FUNCTION_BLOCK FB_Transfo_Base
//////////////////
// High Voltage transformer with Transfo or DMCR detection . 
//////////////////

VAR_INPUT PERSISTENT
	// Parameters of the Object (instance/model specific) 

END_VAR

VAR_OUTPUT
	//Child objects
	
END_VAR

VAR_INPUT
		// Transfo

END_VAR

VAR
	//MesDataExd					: Transfo ; 
		
END_VAR

METHOD M_Execute
//////////////////
//  Method Calls 
/////////////////

VAR 
	// Method local variables (reinitialized at each cycle) 

END_VAR
END_METHOD

END_FUNCTION_BLOCK

(* stored: Version 1.1.0.1, ProductVersion 3.1.4024.6
   POU FB_Transfo_Base: Id {cfe582a0-0c9f-4eac-9b4d-85c949d4eaf5}, SpecialFunc None
   Method M_Execute: Id {3e1fdba9-7259-4a22-9e0e-06ea571a5c31} *)
